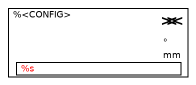
[picture p181: ZLIB_ENCODER_IN (HMI screen)]
rectangle at (0,0)-(180,69): text "%<CONFIG>"; shows $Object$.InstName
rectangle at (8,54)-(173,67): text "%s"; shows $Object$.ErrorString; invisible if $Object$.ErrorString=''
rectangle at (150,27)-(179,41): text "°"
rectangle at (150,40)-(179,54): text "mm"; invisible if $Object$.sInit.lr_LaengeProRpm = 0
group at (149,0)-(179,25)
  rectangle at (0,0)-(30,25): text ">"; invisible if $Object$.Drehrichtung <> 1
  rectangle at (0,0)-(30,25): text "<"; invisible if $Object$.Drehrichtung <> -1
  rectangle at (0,0)-(30,25): text "><"; invisible if $Object$.Drehrichtung <> 0
3 elements of other kinds (tables, trends, ...) not read
*)

(* Visualisation zLibrary/MachineObjects/EsponRobot/ZLIB_EPSON_DETAILS
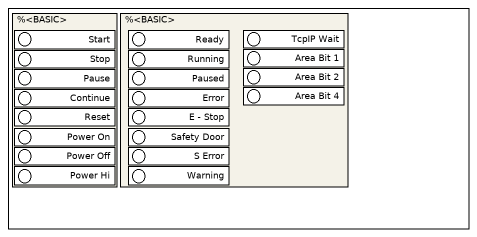
rectangle at (4,5)-(109,179): text "%<BASIC>"; shows 'RoboInput'
rectangle at (112,5)-(340,179): text "%<BASIC>"; shows 'RoboOutput'
rectangle at (6,22)-(107,41): text "Start"
ellipse at (10,24)-(23,38): alarm colour if $Object$.RemOutStart
rectangle at (6,42)-(107,60): text "Stop"
ellipse at (10,44)-(23,58): alarm colour if $Object$.RemOutStop
rectangle at (6,61)-(107,80): text "Pause"
ellipse at (10,63)-(23,77): alarm colour if $Object$.RemOutPause
rectangle at (6,81)-(107,99): text "Continue"
ellipse at (10,83)-(23,97): alarm colour if $Object$.RemOutCont
rectangle at (6,100)-(107,118): text "Reset"
ellipse at (10,102)-(23,116): alarm colour if $Object$.RemOutReset
rectangle at (6,120)-(107,138): text "Power On"
ellipse at (10,122)-(23,136): alarm colour if $Object$.RemOutPowerOn
rectangle at (6,139)-(107,157): text "Power Off"
ellipse at (10,141)-(23,155): alarm colour if $Object$.RemOutPowerOff
rectangle at (6,158)-(107,177): text "Power Hi"
ellipse at (10,161)-(23,175): alarm colour if $Object$.RemOutPowerHi
rectangle at (120,22)-(221,41): text "Ready"
ellipse at (124,24)-(137,38): alarm colour if $Object$.RemInReady
rectangle at (120,42)-(221,60): text "Running"
ellipse at (124,44)-(137,58): alarm colour if $Object$.RemInRunning
rectangle at (120,61)-(221,80): text "Paused"
ellipse at (124,63)-(137,77): alarm colour if $Object$.RemInPaused
rectangle at (120,81)-(221,99): text "Error"
ellipse at (124,83)-(137,97): alarm colour if $Object$.RemInError
rectangle at (120,100)-(221,118): text "E - Stop"
ellipse at (124,102)-(137,116): alarm colour if $Object$.RemInEStopOn
rectangle at (120,120)-(221,138): text "Safety Door"
ellipse at (124,122)-(137,136): alarm colour if $Object$.RemInSafeguardOn
rectangle at (120,139)-(221,157): text "S Error"
ellipse at (124,141)-(137,155): alarm colour if $Object$.RemInSError
rectangle at (120,158)-(221,177): text "Warning"
ellipse at (124,161)-(137,175): alarm colour if $Object$.RemInWarning
rectangle at (235,41)-(336,59): text "Area Bit 1"
ellipse at (239,43)-(252,57): alarm colour if $Object$.RemInAreaBit1
rectangle at (235,60)-(336,78): text "Area Bit 2"
ellipse at (239,62)-(252,76): alarm colour if $Object$.RemInAreaBit2
rectangle at (235,79)-(336,97): text "Area Bit 4"
ellipse at (239,81)-(252,95): alarm colour if $Object$.RemInAreaBit4
rectangle at (235,22)-(336,40): text "TcpIP Wait"
ellipse at (239,24)-(252,38): alarm colour if $Object$.RemInTcpIP_Wait
1 more shapes without text or variables
1 elements of other kinds (tables, trends, ...) not read
*)

(* Visualisation zLibrary/MachineObjects/EsponRobot/ZLIB_EPSON_POSLIST
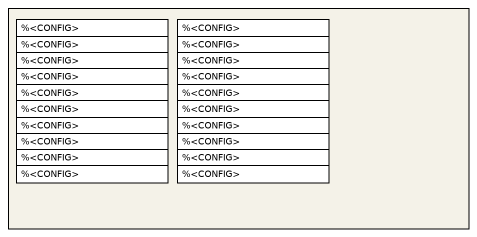
rectangle at (169,11)-(321,29): text "%<CONFIG>"; shows $Object$.PosArray[11]
rectangle at (169,28)-(321,45): text "%<CONFIG>"; shows $Object$.PosArray[12]
rectangle at (169,44)-(321,61): text "%<CONFIG>"; shows $Object$.PosArray[13]
rectangle at (169,60)-(321,77): text "%<CONFIG>"; shows $Object$.PosArray[14]
rectangle at (169,76)-(321,94): text "%<CONFIG>"; shows $Object$.PosArray[15]
rectangle at (169,92)-(321,110): text "%<CONFIG>"; shows $Object$.PosArray[16]
rectangle at (169,109)-(321,126): text "%<CONFIG>"; shows $Object$.PosArray[17]
rectangle at (169,125)-(321,142): text "%<CONFIG>"; shows $Object$.PosArray[18]
rectangle at (169,141)-(321,158): text "%<CONFIG>"; shows $Object$.PosArray[19]
rectangle at (169,157)-(321,175): text "%<CONFIG>"; shows $Object$.PosArray[20]
rectangle at (8,11)-(160,29): text "%<CONFIG>"; shows $Object$.PosArray[1]
rectangle at (8,28)-(160,45): text "%<CONFIG>"; shows $Object$.PosArray[2]
rectangle at (8,44)-(160,61): text "%<CONFIG>"; shows $Object$.PosArray[3]
rectangle at (8,60)-(160,77): text "%<CONFIG>"; shows $Object$.PosArray[4]
rectangle at (8,76)-(160,94): text "%<CONFIG>"; shows $Object$.PosArray[5]
rectangle at (8,92)-(160,110): text "%<CONFIG>"; shows $Object$.PosArray[6]
rectangle at (8,109)-(160,126): text "%<CONFIG>"; shows $Object$.PosArray[7]
rectangle at (8,125)-(160,142): text "%<CONFIG>"; shows $Object$.PosArray[8]
rectangle at (8,141)-(160,158): text "%<CONFIG>"; shows $Object$.PosArray[9]
rectangle at (8,157)-(160,175): text "%<CONFIG>"; shows $Object$.PosArray[10]
1 more shapes without text or variables
1 elements of other kinds (tables, trends, ...) not read
*)

(* Visualisation zLibrary/MachineObjects/EsponRobot/ZLIB_EPSON_ROBOT
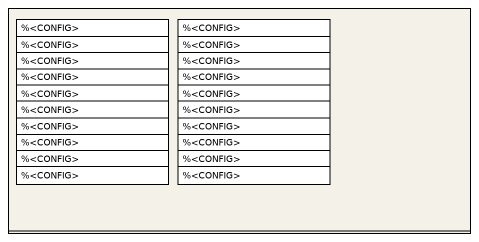
embedded screen at (0,0)-(463,226): ZLIB_EPSON_Steuerung
embedded screen at (0,0)-(463,223): ZLIB_EPSON_DETAILS
embedded screen at (0,0)-(463,223): ZLIB_EPSON_POSLIST
*)

(* Visualisation zLibrary/MachineObjects/EsponRobot/ZLIB_EPSON_STEUERUNG
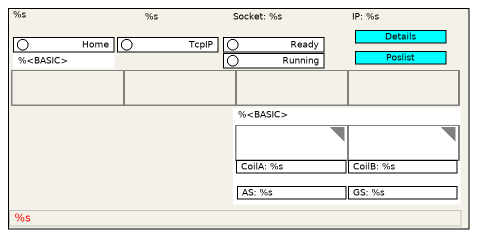
rectangle at (0,0)-(461,221): text "%s"; shows $Object$.BitName
rectangle at (215,29)-(316,44): text "Ready"
ellipse at (219,31)-(230,42): alarm colour if $Object$.RemInReady
rectangle at (215,45)-(316,60): text "Running"
ellipse at (219,47)-(230,58): alarm colour if $Object$.RemInRunning
rectangle at (5,45)-(106,60): text "%d"; shows $Object$.ActualArea
embedded screen at (3,62)-(116,97): ZLIB_VISUBUTTON
rectangle at (1,202)-(453,218): text "%s"; shows $Object$.ErrorString; invisible if $Object$.ErrorPresent
rectangle at (69,2)-(218,15): text "%s"; shows $Object$.Description
embedded screen at (339,62)-(451,97): zLib_VisuButton
embedded screen at (115,62)-(228,97): zLib_VisuButton
embedded screen at (227,62)-(340,97): zLib_VisuButton
rectangle at (5,29)-(106,44): text "Home"
ellipse at (9,31)-(20,42): alarm colour if $Object$.HomePosition
rectangle at (109,29)-(210,44): text "TcpIP"
ellipse at (113,31)-(124,42): alarm colour if $Object$.ConnectionAlive
rectangle at (225,100)-(452,196): text "%<BASIC>"; shows 'Tool'
embedded screen at (227,117)-(340,152): zLib_VisuButton
embedded screen at (339,117)-(451,152): zLib_VisuButton
rectangle at (228,152)-(338,165): text "CoilA: %s"; shows $Object$.NameCoilA; alarm colour if $Object$.RemInToolCoilA
rectangle at (340,152)-(449,165): text "CoilB: %s"; shows $Object$.NameCoilB; invisible if $Object$.NameCoilB='xxxx'; alarm colour if $Object$.RemInToolCoilB
rectangle at (340,178)-(449,191): text "GS: %s"; shows $Object$.NameInitSensor; invisible if $Object$.NameInitSensor='xxxx'; alarm colour if $Object$.RemInToolInitSensor
rectangle at (229,178)-(338,191): text "AS: %s"; shows $Object$.NameWorkSensor; invisible if $Object$.NameWorkSensor='xxxx'; alarm colour if $Object$.RemInToolWorkSensor
rectangle at (339,2)-(452,15): text "IP: %s"; shows $Object$.TcpIpAdress
rectangle at (220,2)-(338,15): text "Socket: %s"; shows $Object$.SocketState
rectangle at (347,43)-(438,56): text "Poslist"; invisible if TRUE
rectangle at (347,22)-(438,35): text "Details"; invisible if TRUE
rectangle at (5,45)-(106,60): text "%<BASIC>"; shows 'ActualArea'
polygon at (322,119)-(336,133): alarm colour if $Object$.RemOutSetToolOn
polygon at (433,119)-(447,133): alarm colour if $Object$.RemOutSetToolOff
12 elements of other kinds (tables, trends, ...) not read
*)

(* Visualisation zLibrary/ErrorHandler/ZLIB_ERRORHANDLER
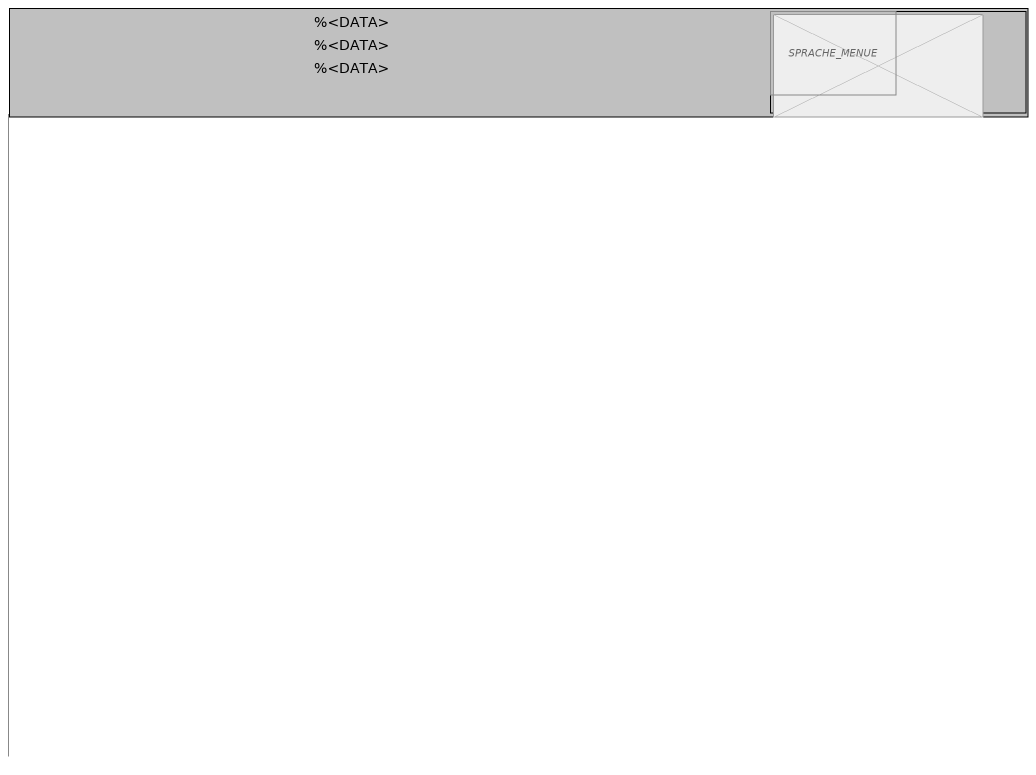
embedded screen at (0,106)-(1017,748): zLib_ErrorList
rectangle at (1,108)-(1020,759): opens ZOOMTOCALLER
bitmap at (765,6)-(975,109): c:\twincat\plc\VisuBmp\ept_logo.jpg
rectangle at (244,27)-(383,47): text "%<DATA>"; shows 'ArtNo'
rectangle at (244,4)-(383,24): text "%<DATA>"; shows 'TypeName'
rectangle at (244,50)-(383,70): text "%<DATA>"; shows 'TypeDescription'
embedded screen at (762,3)-(888,87): SPRACHE_MENUE
2 more shapes without text or variables
4 elements of other kinds (tables, trends, ...) not read
*)

(* Visualisation zLibrary/ErrorHandler/ZLIB_ERRORLINE
3 elements of other kinds (tables, trends, ...) not read
*)

(* Visualisation zLibrary/ErrorHandler/ZLIB_ERRORLIST
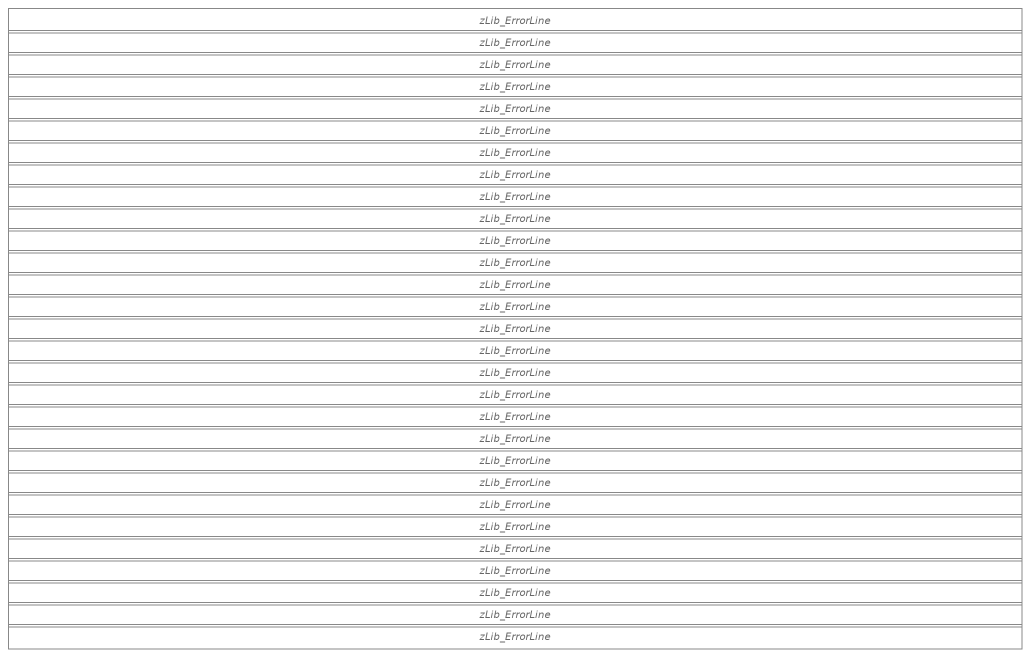
embedded screen at (0,0)-(1014,25): zLib_ErrorLine
embedded screen at (0,22)-(1014,47): zLib_ErrorLine
embedded screen at (0,44)-(1014,69): zLib_ErrorLine
embedded screen at (0,66)-(1014,91): zLib_ErrorLine
embedded screen at (0,88)-(1014,113): zLib_ErrorLine
embedded screen at (0,110)-(1014,135): zLib_ErrorLine
embedded screen at (0,132)-(1014,157): zLib_ErrorLine
embedded screen at (0,154)-(1014,179): zLib_ErrorLine
embedded screen at (0,176)-(1014,201): zLib_ErrorLine
embedded screen at (0,198)-(1014,223): zLib_ErrorLine
embedded screen at (0,220)-(1014,245): zLib_ErrorLine
embedded screen at (0,242)-(1014,267): zLib_ErrorLine
embedded screen at (0,264)-(1014,289): zLib_ErrorLine
embedded screen at (0,286)-(1014,311): zLib_ErrorLine
embedded screen at (0,308)-(1014,333): zLib_ErrorLine
embedded screen at (0,330)-(1014,355): zLib_ErrorLine
embedded screen at (0,352)-(1014,377): zLib_ErrorLine
embedded screen at (0,374)-(1014,399): zLib_ErrorLine
embedded screen at (0,396)-(1014,421): zLib_ErrorLine
embedded screen at (0,418)-(1014,443): zLib_ErrorLine
embedded screen at (0,440)-(1014,465): zLib_ErrorLine
embedded screen at (0,462)-(1014,487): zLib_ErrorLine
embedded screen at (0,484)-(1014,509): zLib_ErrorLine
embedded screen at (0,506)-(1014,531): zLib_ErrorLine
embedded screen at (0,528)-(1014,553): zLib_ErrorLine
embedded screen at (0,550)-(1014,575): zLib_ErrorLine
embedded screen at (0,572)-(1014,597): zLib_ErrorLine
embedded screen at (0,594)-(1014,619): zLib_ErrorLine
embedded screen at (0,616)-(1014,641): zLib_ErrorLine
*)

(* Visualisation zLibrary/ept/ZLIB_IFM
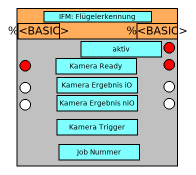
rectangle at (15,110)-(146,129): text "%<BASIC>"; shows 'Kamera Trigger'
rectangle at (15,69)-(146,88): text "%<BASIC>"; shows 'Kamera Ergebnis iO'
rectangle at (15,86)-(146,105): text "%<BASIC>"; shows 'Kamera Ergebnis niO'
ellipse at (147,73)-(158,84): alarm colour if ST02_FDB_56X1_6_IO.BitInToCheck
ellipse at (147,90)-(158,101): alarm colour if ST02_FDB_56X1_6_NIO.BitInToCheck
rectangle at (15,47)-(146,66): text "%<BASIC>"; shows 'Kamera Ready'
ellipse at (147,51)-(158,62): alarm colour if ST02_FDB_56X1_5_READY.BitInToCheck
rectangle at (40,134)-(121,153): text "%<BASIC>"; shows 'Job Nummer'
ellipse at (147,34)-(158,45): alarm colour if MP.ST00.IFMCameraActive
ellipse at (3,74)-(14,85): alarm colour if ST02_FDB_55X1_6_IO.BitInToCheck
ellipse at (3,91)-(14,102): alarm colour if ST02_FDB_55X1_6_NIO.BitInToCheck
ellipse at (3,52)-(14,63): alarm colour if ST02_FDB_55X1_5_READY.BitInToCheck
rectangle at (62,30)-(143,49): text "%<BASIC>"; shows 'aktiv'
rectangle at (0,0)-(161,31): text "%<BASIC>"; shows 'IFM_Flügelerkennung'
rectangle at (1,15)-(43,31): text "%<BASIC>"; shows 'links'
rectangle at (64,33)-(145,49): text "aktiv"; invisible if TRUE
rectangle at (39,50)-(120,66): text "Kamera Ready"; invisible if TRUE
rectangle at (40,69)-(121,85): text "Kamera Ergebnis iO"; invisible if TRUE
rectangle at (40,87)-(121,103): text "Kamera Ergebnis niO"; invisible if TRUE
rectangle at (40,111)-(121,127): text "Kamera Trigger"; invisible if TRUE
rectangle at (42,136)-(123,152): text "Job Nummer"; invisible if TRUE
rectangle at (120,15)-(161,31): text "%<BASIC>"; shows 'rechts'
rectangle at (27,3)-(135,14): text "IFM: Flügelerkennung"; invisible if TRUE
1 more shapes without text or variables
5 elements of other kinds (tables, trends, ...) not read
*)

(* Visualisation zLibrary/MachineObjects/LoginDialog/ZLIB_LOGIN
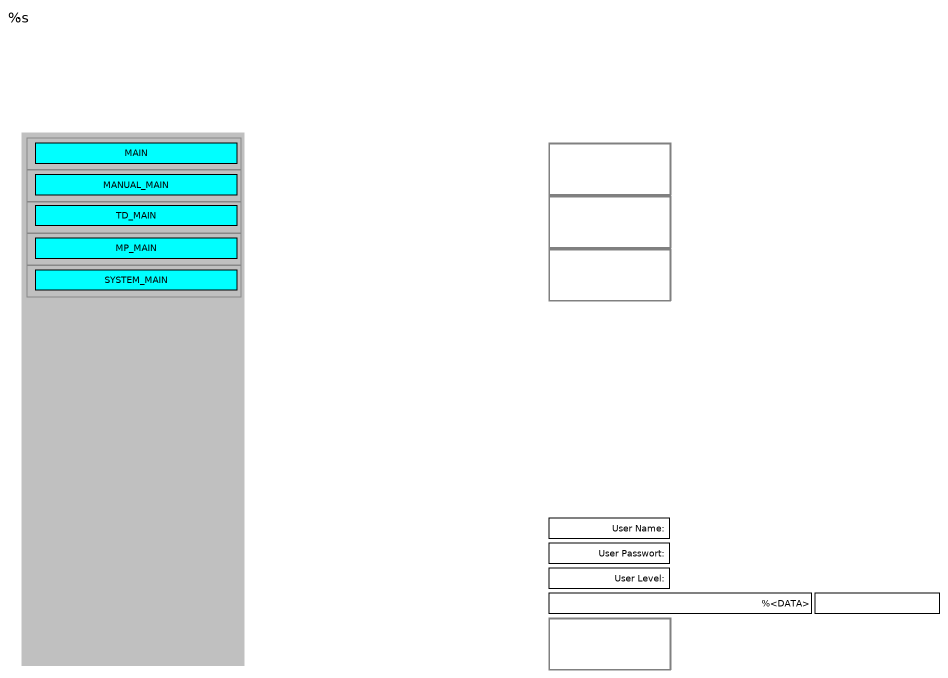
embedded screen at (530,231)-(652,283): ZLIB_VISUBUTTON
rectangle at (0,0)-(0,0): text "%s"; shows UD.UserList[INDEX].UserName; alarm colour if $ROWCONST$ = .Visu.LoginHandler.UserListIndex
embedded screen at (530,125)-(652,177): ZLIB_VISUBUTTON
embedded screen at (530,178)-(652,230): ZLIB_VISUBUTTON
rectangle at (530,500)-(651,521): text "User Name:"; invisible if NOT .Visu.LoginHandler.ShowEditFields
rectangle at (530,575)-(793,596): text "%<DATA>"; shows 'Passwort ändern'; invisible if NOT .Visu.LoginHandler.ShowEditFields
rectangle at (530,525)-(651,546): text "User Passwort:"; invisible if NOT .Visu.LoginHandler.ShowEditFields
rectangle at (530,550)-(651,571): text "User Level:"; invisible if NOT .Visu.LoginHandler.ShowEditFields
rectangle at (796,575)-(921,596): invisible if NOT .Visu.LoginHandler.ShowEditFields; alarm colour if .Visu.LoginHandler.UserEdit.UserCanChangeOwnPassword; toggles .Visu.LoginHandler.UserEdit.UserCanChangeOwnPassword
embedded screen at (530,600)-(652,652): ZLIB_VISUBUTTON
embedded screen at (3,115)-(226,648): M0000_Main
6 elements of other kinds (tables, trends, ...) not read
*)

(* Visualisation zLibrary/MessageHandler/ZLIB_MESSAGELINE
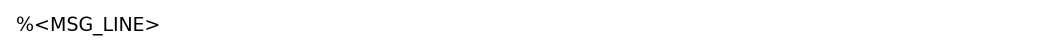
embedded screen at (0,0)-(1025,33): zLib_MessageLineBool
embedded screen at (0,0)-(1025,33): zLib_MessageLineDint
embedded screen at (0,0)-(1025,33): zLib_MessageLineReal
embedded screen at (0,0)-(1025,33): zLib_MessageLineString
*)

(* Visualisation zLibrary/MessageHandler/ZLIB_MESSAGELINEBOOL
rectangle at (0,0)-(969,29): text "%<MSG_LINE>"; shows $MsgLine$.Text; invisible if NOT $MsgLine$.Visible; toggles $MsgLine$.MsgBool
1 elements of other kinds (tables, trends, ...) not read
*)

(* Visualisation zLibrary/MessageHandler/ZLIB_MESSAGELINEDINT
2 elements of other kinds (tables, trends, ...) not read
*)

(* Visualisation zLibrary/MessageHandler/ZLIB_MESSAGELINEREAL
rectangle at (0,0)-(805,29): text "%<MSG_LINE>"; shows $MsgLine$.Text; invisible if NOT $MsgLine$.Visible
1 elements of other kinds (tables, trends, ...) not read
*)

(* Visualisation zLibrary/MessageHandler/ZLIB_MESSAGELINESTRING
rectangle at (0,0)-(805,29): text "%<MSG_LINE>"; shows $MsgLine$.Text; invisible if NOT $MsgLine$.Visible
1 elements of other kinds (tables, trends, ...) not read
*)

(* Visualisation zLibrary/MachineObjects/LoginDialog/ZLIB_NUMERIC_KEYPAD
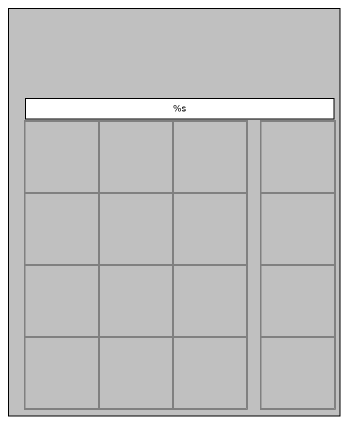
rectangle at (5,4)-(314,25): text "%s"; shows $sNumericKeypad$.InputString
embedded screen at (4,26)-(79,99): ZLIB_VISUBUTTON
embedded screen at (78,26)-(153,99): ZLIB_VISUBUTTON
embedded screen at (152,26)-(227,99): ZLIB_VISUBUTTON
embedded screen at (4,98)-(79,171): ZLIB_VISUBUTTON
embedded screen at (78,98)-(153,171): ZLIB_VISUBUTTON
embedded screen at (152,98)-(227,171): ZLIB_VISUBUTTON
embedded screen at (4,170)-(79,243): ZLIB_VISUBUTTON
embedded screen at (78,170)-(153,243): ZLIB_VISUBUTTON
embedded screen at (152,242)-(227,315): ZLIB_VISUBUTTON
embedded screen at (4,242)-(79,315): ZLIB_VISUBUTTON
embedded screen at (78,242)-(153,315): ZLIB_VISUBUTTON
embedded screen at (152,170)-(227,243): ZLIB_VISUBUTTON
embedded screen at (240,26)-(315,99): ZLIB_VISUBUTTON
embedded screen at (240,98)-(315,171): ZLIB_VISUBUTTON
embedded screen at (240,170)-(315,243): ZLIB_VISUBUTTON
embedded screen at (240,242)-(315,315): ZLIB_VISUBUTTON
1 more shapes without text or variables
*)

(* Visualisation zLibrary/ept/ZLIB_OVERRIDE
rectangle at (0,0)-(101,41): alarm colour if $override$<$overrideVorgabe$
1 more shapes without text or variables
3 elements of other kinds (tables, trends, ...) not read
*)

(* Visualisation zLibrary/ept/ZLIB_SCHWENKARM
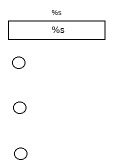
rectangle at (0,0)-(101,171): text "%s"; shows '$FB$'
rectangle at (2,13)-(99,32): text "%s"; shows $FB$.fb_state_entry.i16_step; alarm colour if $FB$.fb_state_entry.i16_step=1000
ellipse at (6,49)-(19,61): alarm colour if $FB$.ST02_90_0_sens
ellipse at (7,94)-(20,106): alarm colour if $FB$.ST02_90_sens
ellipse at (8,140)-(21,152): alarm colour if $FB$.ST02_90_180_sens
6 elements of other kinds (tables, trends, ...) not read
*)

(* Visualisation zLibrary/ept/Sensopart/ZLIB_SENSOPART
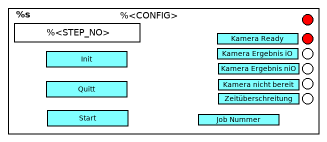
rectangle at (0,0)-(311,126): text "%s"; shows '$FB$'
rectangle at (178,21)-(289,40): text "%<BASIC>"; shows 'Kamera Ready'
rectangle at (178,36)-(289,55): text "%<BASIC>"; shows 'Kamera Ergebnis iO'
rectangle at (178,51)-(289,70): text "%<BASIC>"; shows 'Kamera Ergebnis niO'
rectangle at (6,15)-(132,34): text "%<STEP_NO>"; shows $FB$.fb_state_entry.i16_step; alarm colour if $FB$.fb_state_entry.i16_step=1000
ellipse at (294,25)-(305,36): alarm colour if $FB$.b_ready
ellipse at (294,40)-(305,51): alarm colour if $FB$.Ergebnis_IO
ellipse at (294,55)-(305,66): alarm colour if $FB$.Ergebnis_NIO
rectangle at (178,66)-(289,85): text "%<BASIC>"; shows 'Kamera nicht betriebsbereit'
ellipse at (294,70)-(305,81): alarm colour if $FB$.sm_kamera_nicht_bb
rectangle at (178,81)-(289,100): text "%<BASIC>"; shows 'Zeitüberschreitung'
ellipse at (294,85)-(305,96): alarm colour if $FB$.sm_zeitueberschreitung
rectangle at (155,104)-(266,123): text "%<BASIC>"; shows 'Job Nummer'
ellipse at (294,6)-(305,17): alarm colour if $Cam_On$
rectangle at (110,1)-(240,14): text "%<CONFIG>"; shows '$FB$'
rectangle at (209,25)-(290,36): text "Kamera Ready"; invisible if TRUE
rectangle at (209,40)-(290,51): text "Kamera Ergebnis iO"; invisible if TRUE
rectangle at (210,55)-(291,66): text "Kamera Ergebnis niO"; invisible if TRUE
rectangle at (210,71)-(291,82): text "Kamera nicht bereit"; invisible if TRUE
rectangle at (210,85)-(291,96): text "Zeitüberschreitung"; invisible if TRUE
rectangle at (190,106)-(271,117): text "Job Nummer"; invisible if TRUE
rectangle at (39,102)-(120,118): text "Start"; invisible if TRUE
rectangle at (38,73)-(119,89): text "Quitt"; invisible if TRUE
rectangle at (38,43)-(119,59): text "Init"; invisible if TRUE
8 elements of other kinds (tables, trends, ...) not read
*)

(* Visualisation zLibrary/ept/Sensopart/ZLIB_SENSOPART_1
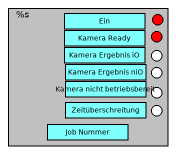
rectangle at (0,0)-(160,138): text "%s"; shows '$FB$'
rectangle at (27,17)-(138,36): text "%<BASIC>"; shows 'Kamera Ready'
rectangle at (27,37)-(138,56): text "%<BASIC>"; shows 'Kamera Ergebnis iO'
rectangle at (27,54)-(138,73): text "%<BASIC>"; shows 'Kamera Ergebnis niO'
ellipse at (143,23)-(154,34): alarm colour if $FB$.b_ready
ellipse at (143,42)-(154,53): alarm colour if $FB$.Ergebnis_IO
ellipse at (143,59)-(154,70): alarm colour if $FB$.Ergebnis_NIO
rectangle at (3,73)-(140,92): text "%<BASIC>"; shows 'Kamera nicht betriebsbereit'
ellipse at (143,79)-(154,90): alarm colour if $FB$.sm_kamera_nicht_bb
rectangle at (27,92)-(138,111): text "%<BASIC>"; shows 'Zeitüberschreitung'
ellipse at (143,97)-(154,108): alarm colour if $FB$.sm_zeitueberschreitung
rectangle at (10,114)-(121,133): text "%<BASIC>"; shows 'Job Nummer'
ellipse at (144,6)-(155,17): alarm colour if $Cam_On$
rectangle at (113,2)-(139,21): text "%<BASIC>"; shows 'Ein'
rectangle at (56,5)-(137,21): text "Ein"; invisible if TRUE
rectangle at (56,22)-(137,38): text "Kamera Ready"; invisible if TRUE
rectangle at (56,39)-(137,55): text "Kamera Ergebnis iO"; invisible if TRUE
rectangle at (57,56)-(138,72): text "Kamera Ergebnis niO"; invisible if TRUE
rectangle at (57,73)-(138,89): text "Kamera nicht betriebsbereit"; invisible if TRUE
rectangle at (57,94)-(138,110): text "Zeitüberschreitung"; invisible if TRUE
rectangle at (39,116)-(120,132): text "Job Nummer"; invisible if TRUE
1 elements of other kinds (tables, trends, ...) not read
*)

(* Visualisation zLibrary/ept/Sensopart/ZLIB_SENSOPART_2
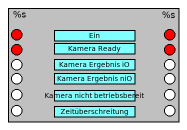
rectangle at (0,0)-(171,114): text "%s"; shows '$FB1$'
ellipse at (156,36)-(167,47): alarm colour if $FB2$.b_ready
ellipse at (156,51)-(167,62): alarm colour if $FB2$.Ergebnis_IO
ellipse at (156,65)-(167,76): alarm colour if $FB2$.Ergebnis_NIO
ellipse at (156,81)-(167,92): alarm colour if $FB2$.sm_kamera_nicht_bb
ellipse at (156,97)-(167,108): alarm colour if $FB2$.sm_zeitueberschreitung
ellipse at (156,21)-(167,32): alarm colour if $Cam_On2$
ellipse at (3,36)-(14,47): alarm colour if $FB1$.b_ready
ellipse at (3,51)-(14,62): alarm colour if $FB1$.Ergebnis_IO
ellipse at (3,65)-(14,76): alarm colour if $FB1$.Ergebnis_NIO
ellipse at (3,81)-(14,92): alarm colour if $FB1$.sm_kamera_nicht_bb
ellipse at (3,97)-(14,108): alarm colour if $FB1$.sm_zeitueberschreitung
ellipse at (3,21)-(14,32): alarm colour if $Cam_On1$
rectangle at (85,0)-(169,14): text "%s"; shows '$FB2$'
rectangle at (17,31)-(154,50): text "%<BASIC>"; shows 'Kamera Ready'
rectangle at (17,47)-(154,66): text "%<BASIC>"; shows 'Kamera Ergebnis iO'
rectangle at (17,61)-(154,80): text "%<BASIC>"; shows 'Kamera Ergebnis niO'
rectangle at (17,77)-(154,96): text "%<BASIC>"; shows 'Kamera nicht betriebsbereit'
rectangle at (17,93)-(154,112): text "%<BASIC>"; shows 'Zeitüberschreitung'
rectangle at (17,18)-(154,37): text "%<BASIC>"; shows 'Ein'
rectangle at (46,22)-(127,33): text "Ein"; invisible if TRUE
rectangle at (46,35)-(127,46): text "Kamera Ready"; invisible if TRUE
rectangle at (46,51)-(127,62): text "Kamera Ergebnis iO"; invisible if TRUE
rectangle at (46,65)-(127,76): text "Kamera Ergebnis niO"; invisible if TRUE
rectangle at (46,82)-(127,93): text "Kamera nicht betriebsbereit"; invisible if TRUE
rectangle at (46,98)-(127,109): text "Zeitüberschreitung"; invisible if TRUE
*)

(* Visualisation zLibrary/ept/Sensopart/ZLIB_SENSOPART_3
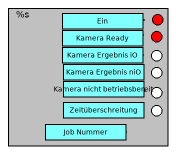
rectangle at (0,0)-(160,138): text "%s"; shows '$FB$'
ellipse at (143,23)-(154,34): alarm colour if $FB$.b_ready
ellipse at (143,42)-(154,53): alarm colour if $FB$.Ergebnis_IO
ellipse at (143,59)-(154,70): alarm colour if $FB$.Ergebnis_NIO
ellipse at (143,79)-(154,90): alarm colour if $FB$.sm_kamera_nicht_bb
ellipse at (143,97)-(154,108): alarm colour if $FB$.sm_zeitueberschreitung
ellipse at (144,6)-(155,17): alarm colour if $Cam_On$
rectangle at (28,17)-(139,36): text "%<BASIC>"; shows 'Kamera Ready'
rectangle at (28,37)-(139,56): text "%<BASIC>"; shows 'Kamera Ergebnis iO'
rectangle at (28,54)-(139,73): text "%<BASIC>"; shows 'Kamera Ergebnis niO'
rectangle at (4,73)-(141,92): text "%<BASIC>"; shows 'Kamera nicht betriebsbereit'
rectangle at (28,92)-(139,111): text "%<BASIC>"; shows 'Zeitüberschreitung'
rectangle at (11,114)-(122,133): text "%<BASIC>"; shows 'Job Nummer'
rectangle at (114,2)-(140,21): text "%<BASIC>"; shows 'Ein'
rectangle at (54,5)-(135,21): text "Ein"; invisible if TRUE
rectangle at (54,22)-(135,38): text "Kamera Ready"; invisible if TRUE
rectangle at (54,39)-(135,55): text "Kamera Ergebnis iO"; invisible if TRUE
rectangle at (55,56)-(136,72): text "Kamera Ergebnis niO"; invisible if TRUE
rectangle at (55,73)-(136,89): text "Kamera nicht betriebsbereit"; invisible if TRUE
rectangle at (55,94)-(136,110): text "Zeitüberschreitung"; invisible if TRUE
rectangle at (37,116)-(118,132): text "Job Nummer"; invisible if TRUE
1 elements of other kinds (tables, trends, ...) not read
*)

(* Visualisation zLibrary/ept/Sensopart/ZLIB_SENSOPART_4
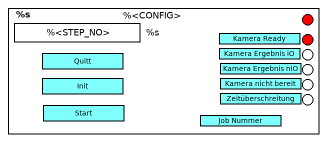
rectangle at (0,0)-(311,126): text "%s"; shows '$FB$'
rectangle at (6,15)-(132,34): text "%<STEP_NO>"; shows $FB$.fb_state_entry.i16_step; alarm colour if $FB$.fb_state_entry.i16_step=1000
ellipse at (294,26)-(305,37): alarm colour if $FB$.st_ctrl_out.b_bereit
ellipse at (294,41)-(305,52): alarm colour if $FB$.b_Kam_Pruef_IO
ellipse at (294,56)-(305,67): alarm colour if $FB$.b_Kam_Pruef_NIO
ellipse at (294,71)-(305,82): alarm colour if $FB$.sm_kamera_nicht_bb
ellipse at (294,86)-(305,97): alarm colour if $FB$.sm_kamera_keine_reaktion
ellipse at (294,6)-(305,17): alarm colour if $Cam_On$
rectangle at (107,1)-(246,14): text "%<CONFIG>"; shows '$FB$'
rectangle at (35,97)-(116,113): text "Start"; invisible if TRUE
rectangle at (34,45)-(115,61): text "Quitt"; invisible if TRUE
rectangle at (34,70)-(115,86): text "Init"; invisible if TRUE
rectangle at (179,22)-(290,41): text "%<BASIC>"; shows 'Kamera Ready'
rectangle at (179,37)-(290,56): text "%<BASIC>"; shows 'Kamera Ergebnis iO'
rectangle at (179,52)-(290,71): text "%<BASIC>"; shows 'Kamera Ergebnis niO'
rectangle at (179,67)-(290,86): text "%<BASIC>"; shows 'Kamera nicht betriebsbereit'
rectangle at (179,82)-(290,101): text "%<BASIC>"; shows 'Zeitüberschreitung'
rectangle at (159,104)-(270,123): text "%<BASIC>"; shows 'Job Nummer'
rectangle at (211,25)-(292,36): text "Kamera Ready"; invisible if TRUE
rectangle at (211,40)-(292,51): text "Kamera Ergebnis iO"; invisible if TRUE
rectangle at (212,55)-(293,66): text "Kamera Ergebnis niO"; invisible if TRUE
rectangle at (212,70)-(293,81): text "Kamera nicht bereit"; invisible if TRUE
rectangle at (212,85)-(293,96): text "Zeitüberschreitung"; invisible if TRUE
rectangle at (192,107)-(273,118): text "Job Nummer"; invisible if TRUE
rectangle at (133,15)-(214,34): text "%s"; shows $FB$.RecvDataString
8 elements of other kinds (tables, trends, ...) not read
*)

(* Visualisation zLibrary/ept/Sensopart/ZLIB_SENSOPART_4_2
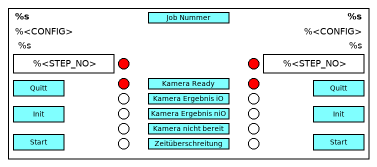
rectangle at (5,46)-(106,65): text "%<STEP_NO>"; shows $FB$.fb_state_entry.i16_step; alarm colour if $FB$.fb_state_entry.i16_step=1000
ellipse at (240,70)-(251,81): alarm colour if $FB2$.st_ctrl_out.b_bereit
ellipse at (240,85)-(251,96): alarm colour if $FB2$.b_Kam_Pruef_IO
ellipse at (240,100)-(251,111): alarm colour if $FB2$.b_Kam_Pruef_NIO
ellipse at (240,115)-(251,126): alarm colour if $FB2$.sm_kamera_nicht_bb
ellipse at (240,130)-(251,141): alarm colour if $FB2$.sm_zeitueberschreitung
ellipse at (240,50)-(251,61): alarm colour if $Cam_On2$
rectangle at (5,17)-(144,30): text "%<CONFIG>"; shows '$FB$'
rectangle at (5,126)-(56,142): text "Start"; invisible if TRUE
rectangle at (5,72)-(56,88): text "Quitt"; invisible if TRUE
rectangle at (5,98)-(56,114): text "Init"; invisible if TRUE
rectangle at (125,66)-(236,85): text "%<BASIC>"; shows 'Kamera Ready'
rectangle at (125,81)-(236,100): text "%<BASIC>"; shows 'Kamera Ergebnis iO'
rectangle at (125,96)-(236,115): text "%<BASIC>"; shows 'Kamera Ergebnis niO'
rectangle at (125,111)-(236,130): text "%<BASIC>"; shows 'Kamera nicht betriebsbereit'
rectangle at (125,126)-(236,145): text "%<BASIC>"; shows 'Zeitüberschreitung'
rectangle at (125,2)-(236,15): text "%<BASIC>"; shows 'Job Nummer'
rectangle at (140,70)-(221,81): text "Kamera Ready"; invisible if TRUE
rectangle at (140,85)-(221,96): text "Kamera Ergebnis iO"; invisible if TRUE
rectangle at (140,100)-(221,111): text "Kamera Ergebnis niO"; invisible if TRUE
rectangle at (140,115)-(221,126): text "Kamera nicht bereit"; invisible if TRUE
rectangle at (140,130)-(221,141): text "Zeitüberschreitung"; invisible if TRUE
rectangle at (140,4)-(221,15): text "Job Nummer"; invisible if TRUE
rectangle at (5,31)-(86,44): text "%s"; shows $FB$.RecvDataString
ellipse at (110,70)-(121,81): alarm colour if $FB$.st_ctrl_out.b_bereit
ellipse at (110,85)-(121,96): alarm colour if $FB$.b_Kam_Pruef_IO
ellipse at (110,100)-(121,111): alarm colour if $FB$.b_Kam_Pruef_NIO
ellipse at (110,115)-(121,126): alarm colour if $FB$.sm_kamera_nicht_bb
ellipse at (110,130)-(121,141): alarm colour if $FB$.sm_zeitueberschreitung
ellipse at (110,50)-(121,61): alarm colour if $Cam_On$
rectangle at (5,2)-(144,15): text "%s"; shows '$FB$'
rectangle at (217,17)-(356,30): text "%<CONFIG>"; shows '$FB2$'
rectangle at (217,2)-(356,15): text "%s"; shows '$FB2$'
rectangle at (275,31)-(356,44): text "%s"; shows $FB2$.RecvDataString
rectangle at (255,46)-(356,65): text "%<STEP_NO>"; shows $FB2$.fb_state_entry.i16_step; alarm colour if $FB2$.fb_state_entry.i16_step=1000
rectangle at (305,126)-(356,142): text "Start"; invisible if TRUE
rectangle at (305,72)-(356,88): text "Quitt"; invisible if TRUE
rectangle at (305,98)-(356,114): text "Init"; invisible if TRUE
1 more shapes without text or variables
16 elements of other kinds (tables, trends, ...) not read
*)

(* Visualisation zLibrary/ept/Sensopart/ZLIB_SENSOPART_5
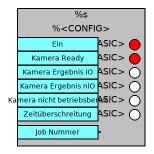
rectangle at (0,0)-(128,138): text "%s"; shows '$FB$'
rectangle at (2,40)-(110,59): text "%<BASIC>"; shows 'Kamera Ready'
rectangle at (2,54)-(110,73): text "%<BASIC>"; shows 'Kamera Ergebnis iO'
rectangle at (2,68)-(110,87): text "%<BASIC>"; shows 'Kamera Ergebnis niO'
rectangle at (2,96)-(110,115): text "%<BASIC>"; shows 'Zeitüberschreitung'
rectangle at (2,114)-(87,133): text "%<BASIC>"; shows 'Job Nummer'
ellipse at (112,31)-(123,42): alarm colour if $Cam_On$
rectangle at (2,26)-(110,45): text "%<BASIC>"; shows 'Ein'
rectangle at (0,29)-(81,43): text "Ein"; invisible if TRUE
rectangle at (0,117)-(81,131): text "Job Nummer"; invisible if TRUE
ellipse at (112,45)-(123,56): alarm colour if $FB$.st_ctrl_out.b_bereit
ellipse at (112,59)-(123,70): alarm colour if $FB$.b_Kam_Pruef_IO
ellipse at (112,73)-(123,84): alarm colour if $FB$.b_Kam_Pruef_NIO
ellipse at (112,87)-(123,98): alarm colour if $FB$.sm_kamera_nicht_bb
ellipse at (112,101)-(123,112): alarm colour if $FB$.sm_zeitueberschreitung
rectangle at (0,43)-(81,57): text "Kamera Ready"; invisible if TRUE
rectangle at (0,57)-(81,71): text "Kamera Ergebnis iO"; invisible if TRUE
rectangle at (0,71)-(81,85): text "Kamera Ergebnis niO"; invisible if TRUE
rectangle at (0,99)-(81,113): text "Zeitüberschreitung"; invisible if TRUE
rectangle at (2,82)-(110,101): text "%<BASIC>"; shows 'Kamera nicht betriebsbereit'
rectangle at (0,85)-(81,99): text "Kamera nicht betriebsbereit"; invisible if TRUE
rectangle at (2,14)-(126,27): text "%<CONFIG>"; shows '$FB$'
1 elements of other kinds (tables, trends, ...) not read
*)

(* Visualisation zLibrary/ept/Sensopart/ZLIB_SENSOPART_6
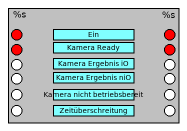
rectangle at (0,0)-(171,115): text "%s"; shows '$FB1$'
rectangle at (16,30)-(153,49): text "%<BASIC>"; shows 'Kamera Ready'
rectangle at (16,46)-(153,65): text "%<BASIC>"; shows 'Kamera Ergebnis iO'
rectangle at (16,60)-(153,79): text "%<BASIC>"; shows 'Kamera Ergebnis niO'
ellipse at (156,36)-(167,47): alarm colour if $FB2$.st_ctrl_out.b_bereit
ellipse at (156,51)-(167,62): alarm colour if $FB2$.b_Kam_Pruef_IO
ellipse at (156,65)-(167,76): alarm colour if $FB2$.b_Kam_Pruef_NIO
rectangle at (16,76)-(153,95): text "%<BASIC>"; shows 'Kamera nicht betriebsbereit'
ellipse at (156,81)-(167,92): alarm colour if $FB2$.sm_kamera_nicht_bb
rectangle at (16,92)-(153,111): text "%<BASIC>"; shows 'Zeitüberschreitung'
ellipse at (156,97)-(167,108): alarm colour if $FB2$.sm_zeitueberschreitung
ellipse at (156,21)-(167,32): alarm colour if $Cam_On2$
rectangle at (16,17)-(153,36): text "%<BASIC>"; shows 'Ein'
ellipse at (3,36)-(14,47): alarm colour if $FB1$.st_ctrl_out.b_bereit
ellipse at (3,51)-(14,62): alarm colour if $FB1$.b_Kam_Pruef_IO
ellipse at (3,65)-(14,76): alarm colour if $FB1$.b_Kam_Pruef_NIO
ellipse at (3,81)-(14,92): alarm colour if $FB1$.sm_kamera_nicht_bb
ellipse at (3,97)-(14,108): alarm colour if $FB1$.sm_zeitueberschreitung
ellipse at (3,21)-(14,32): alarm colour if $Cam_On1$
rectangle at (85,0)-(169,14): text "%s"; shows '$FB2$'
rectangle at (45,21)-(126,32): text "Ein"; invisible if TRUE
rectangle at (45,34)-(126,45): text "Kamera Ready"; invisible if TRUE
rectangle at (45,50)-(126,61): text "Kamera Ergebnis iO"; invisible if TRUE
rectangle at (45,64)-(126,75): text "Kamera Ergebnis niO"; invisible if TRUE
rectangle at (45,81)-(126,92): text "Kamera nicht betriebsbereit"; invisible if TRUE
rectangle at (45,97)-(126,108): text "Zeitüberschreitung"; invisible if TRUE
*)

(* Visualisation zLibrary/ept/Sensopart/ZLIB_SENSOPART_7
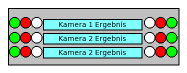
rectangle at (34,5)-(134,24): text "%<BASIC>"; shows 'Kamera 1 Ergebnis'
rectangle at (34,19)-(134,38): text "%<BASIC>"; shows 'Kamera 2 Ergebnis'
ellipse at (147,24)-(158,35): alarm colour if $FB2$.st_ctrl_out.b_bereit
ellipse at (136,9)-(147,20): alarm colour if $FB2$.b_Kam_Pruef_IO
ellipse at (136,24)-(147,35): alarm colour if $FB2$.b_Kam_Pruef_NIO
ellipse at (136,38)-(147,49): alarm colour if $FB2$.sm_kamera_nicht_bb
ellipse at (147,9)-(158,20): alarm colour if $Cam_On2$
ellipse at (12,24)-(23,35): alarm colour if $FB1$.st_ctrl_out.b_bereit
ellipse at (23,9)-(34,20): alarm colour if $FB1$.b_Kam_Pruef_IO
ellipse at (23,24)-(34,35): alarm colour if $FB1$.b_Kam_Pruef_NIO
ellipse at (23,38)-(34,49): alarm colour if $FB1$.sm_kamera_nicht_bb
ellipse at (12,9)-(23,20): alarm colour if $Cam_On1$
rectangle at (34,33)-(134,52): text "%<BASIC>"; shows 'Kamera 3 Ergebnis'
ellipse at (147,38)-(158,49): alarm colour if $FB2$.st_ctrl_out.b_bereit
ellipse at (12,38)-(23,49): alarm colour if $FB1$.st_ctrl_out.b_bereit
ellipse at (158,24)-(169,35): alarm colour if $FB2$.st_ctrl_out.b_bereit
ellipse at (158,9)-(169,20): alarm colour if $Cam_On2$
ellipse at (158,38)-(169,49): alarm colour if $FB2$.st_ctrl_out.b_bereit
ellipse at (1,24)-(12,35): alarm colour if $FB2$.st_ctrl_out.b_bereit
ellipse at (1,9)-(12,20): alarm colour if $Cam_On2$
ellipse at (1,38)-(12,49): alarm colour if $FB2$.st_ctrl_out.b_bereit
rectangle at (35,11)-(134,22): text "Kamera 1 Ergebnis"; invisible if TRUE
rectangle at (35,25)-(134,36): text "Kamera 2 Ergebnis"; invisible if TRUE
rectangle at (35,39)-(134,50): text "Kamera 2 Ergebnis"; invisible if TRUE
1 more shapes without text or variables
*)

(* Visualisation zLibrary/MachineObjects/DigIn/ZLIB_SENSORCHECK
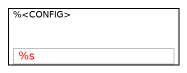
rectangle at (0,0)-(171,57): text "%<CONFIG>"; shows $Object$.InstName
rectangle at (5,40)-(166,56): text "%s"; shows $Object$.ErrorString; invisible if NOT $Object$.ErrorPresent
2 elements of other kinds (tables, trends, ...) not read
*)

(* Visualisation zLibrary/VisuObjects/SERVICE/ZLIB_SERVICELINE
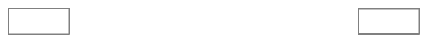
embedded screen at (355,0)-(416,26): ZLIB_VISUBUTTON_TOGGELN
embedded screen at (705,0)-(766,26): ZLIB_VISUBUTTON
embedded screen at (705,0)-(766,26): ZLIB_VISUBUTTON_S17
8 elements of other kinds (tables, trends, ...) not read
*)

(* Visualisation zLibrary/VisuObjects/SERVICE/ZLIB_SERVICELIST
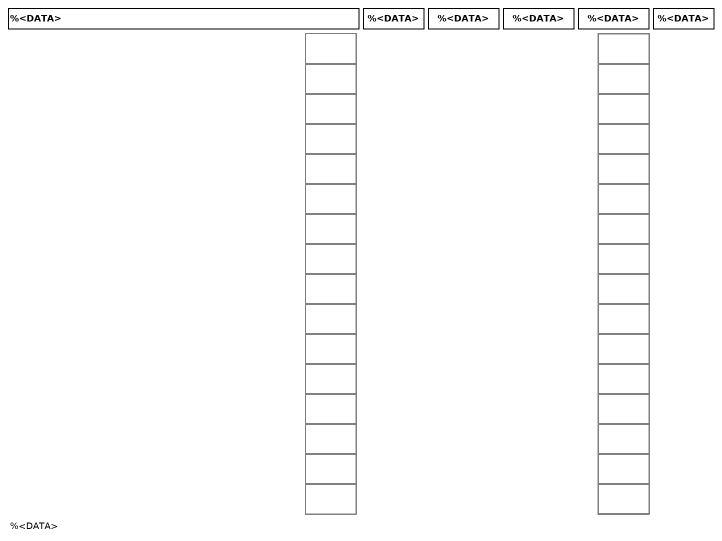
embedded screen at (0,25)-(641,56): ZLIB_SERVICELINE
embedded screen at (0,55)-(641,86): ZLIB_SERVICELINE
rectangle at (0,0)-(351,21): text "%<DATA>"; shows 'Bezeichung der Wartung'
rectangle at (355,0)-(416,21): text "%<DATA>"; shows 'Art'
rectangle at (420,0)-(491,21): text "%<DATA>"; shows 'Vorgabe'
rectangle at (495,0)-(566,21): text "%<DATA>"; shows 'Warngrenze'
rectangle at (570,0)-(641,21): text "%<DATA>"; shows 'Aktuell'
rectangle at (645,0)-(706,21): text "%<DATA>"; shows 'Einheit'
embedded screen at (0,85)-(641,116): ZLIB_SERVICELINE
embedded screen at (0,115)-(641,146): ZLIB_SERVICELINE
embedded screen at (0,145)-(641,176): ZLIB_SERVICELINE
embedded screen at (0,175)-(641,206): ZLIB_SERVICELINE
embedded screen at (0,205)-(641,236): ZLIB_SERVICELINE
embedded screen at (0,235)-(641,266): ZLIB_SERVICELINE
embedded screen at (0,265)-(641,296): ZLIB_SERVICELINE
embedded screen at (0,295)-(641,326): ZLIB_SERVICELINE
embedded screen at (0,325)-(641,356): ZLIB_SERVICELINE
embedded screen at (0,355)-(641,386): ZLIB_SERVICELINE
embedded screen at (0,385)-(641,416): ZLIB_SERVICELINE
embedded screen at (0,415)-(641,446): ZLIB_SERVICELINE
embedded screen at (0,445)-(641,476): ZLIB_SERVICELINE
embedded screen at (0,475)-(641,506): ZLIB_SERVICELINE
rectangle at (0,505)-(766,531): text "%<DATA>"; shows 'Info'
*)

(* Visualisation zLibrary/VisuObjects/ZLIB_SFC_STATE
